TYPE "SpeedMachine_Wng"
VERSION : 0.1
// Block: SpeedMachine_Wng
   STRUCT
      NotAutReady : Bool;
      MissingCnd_Bkw : Bool;
      MissingCnd_Fwd : Bool;
      Ax : Struct
         Drive : Bool;
      END_STRUCT;
   END_STRUCT;

END_TYPE
